// TIA Portal V17 export
// export: Created 2025-03-11T12:28:51.4974891Z, ExportSetting WithDefaults, DisplayName Totally Integrated Automation Portal, DisplayVersion V17 Update 8, DisplayName TIA Portal Openness, DisplayVersion V17 Update 8, DisplayName TIA Portal Version Control Interface, DisplayVersion V17, DisplayName SINAMICS Startdrive Advanced, DisplayVersion V17 SP2, DisplayName SINAMICS Startdrive G110M, G120, G120C, G120D, G120P, G115D, DisplayVersion V17 SP2, DisplayName SINAMICS Startdrive G130, G150, S120, S150, SINAMICS MV, S210, DisplayVersion V17 SP2, DisplayName STEP 7 Professional, DisplayVersion V17 Update 8, DisplayName SINUMERIK ONE STEP 7 Toolbox, DisplayVersion V17 Update 12, DisplayName SINUMERIK 840D sl STEP 7 Toolbox, DisplayVersion V17 Update 12, DisplayName STEP 7 Safety, DisplayVersion V17 Update 6, DisplayName WinCC Advanced, DisplayVersion V17 Update 8
DATA_BLOCK "DB21222_POWDER_FILLING_START_STOP_BY_CURRENT_DB"   // DB21222
{ DB_Accessible_From_OPC_UA := 'FALSE' }
VERSION : 0.1
// stored: AutoNumber false, DBAccessibleFromOPCUA false, DBAccessibleFromWebserver true, InstanceOfName FB21222_POWDER_FILLING_START_STOP_BY_CURRENT, InstanceOfType FB
"FB21222_POWDER_FILLING_START_STOP_BY_CURRENT"
   // VAR_INPUT
   //    SENSOR_VALUE : Int;
   //    iFEEDER_STATE_LINE : Word;
   //    HMI_HIGH_CURRENT_LIMIT : Real;
   //    HMI_LOW_CURRENT_LIMIT : Real;
   // END_VAR
   // VAR_OUTPUT
   //    POWDER_FILLING_STOP_BY_CURRENT : Bool;
   //    POWDER_FILLING_START_BY_CURRENT : Bool;
   // END_VAR
   // VAR
   //    CURRENT_AVG_BLCK_START : Real;
   //    CURRENT_AVG_BLCK_STOP : Real;
   //    CURRENT_AVG_BLCK_HMI_START : Real;
   //    CURRENT_AVG_BLCK_HMI_STOP : Real;
   //    PF_LINE_ON : Bool;
   //    NORMALIZED_VALUE : Real;
   //    SCALED_VALUE : Real;
   //    DB_CURRENT_AVERAGE_START : "FB21990_LGF_FloatingAverage";
   //    DB_CURRENT_AVERAGE_STOP { S7_SetPoint := 'True'} : "FB21990_LGF_FloatingAverage";
   //    TON_TIME { S7_SetPoint := 'True'} : TON_TIME;
   // END_VAR
BEGIN
END_DATA_BLOCK
